TYPE SValue :
STRUCT
	DataType: EDataType;
	Value: UValues;
	Defined: BOOL;
END_STRUCT
END_TYPE

(* stored: Version 1.1.0.1, ProductVersion 3.1.4024.9
   DUT SValue: Id {96b85e64-68fa-4318-bae9-2420a9e5267f} *)
